// TIA Portal V16 export
// export: Created 2022-11-17T11:55:06.396Z, ExportSetting WithDefaults, DisplayName Totally Integrated Automation Portal, DisplayVersion V16 Update 6, DisplayName TIA Portal Version Control Interface, DisplayVersion V16 Update 2, DisplayName TIA Portal Openness, DisplayVersion V16 Update 6, DisplayName SINAMICS Startdrive Advanced, DisplayVersion V16 Update 5, DisplayName SINAMICS Startdrive G130, G150, S120, S150, SINAMICS MV, S210, DisplayVersion V16 Update 5, DisplayName SINAMICS Startdrive G110M, G120, G120C, G120D, G120P, G115D, DisplayVersion V16 Update 5, DisplayName STEP 7 Professional, DisplayVersion V16 Update 6, DisplayName STEP 7 Safety, DisplayVersion V16, DisplayName WinCC Advanced, DisplayVersion V16 Update 6
FUNCTION "FC11_PressureRectangularPn5W" : Void   // FC11, LAD
{ S7_Optimized_Access := 'FALSE' }
VERSION : 0.1
// stored: AutoNumber false, IsIECCheckEnabled false, SetENOAutomatically false, UDAEnableTagReadback false
BEGIN

REGION Network 1: Timeout for pressure plate upward/downward
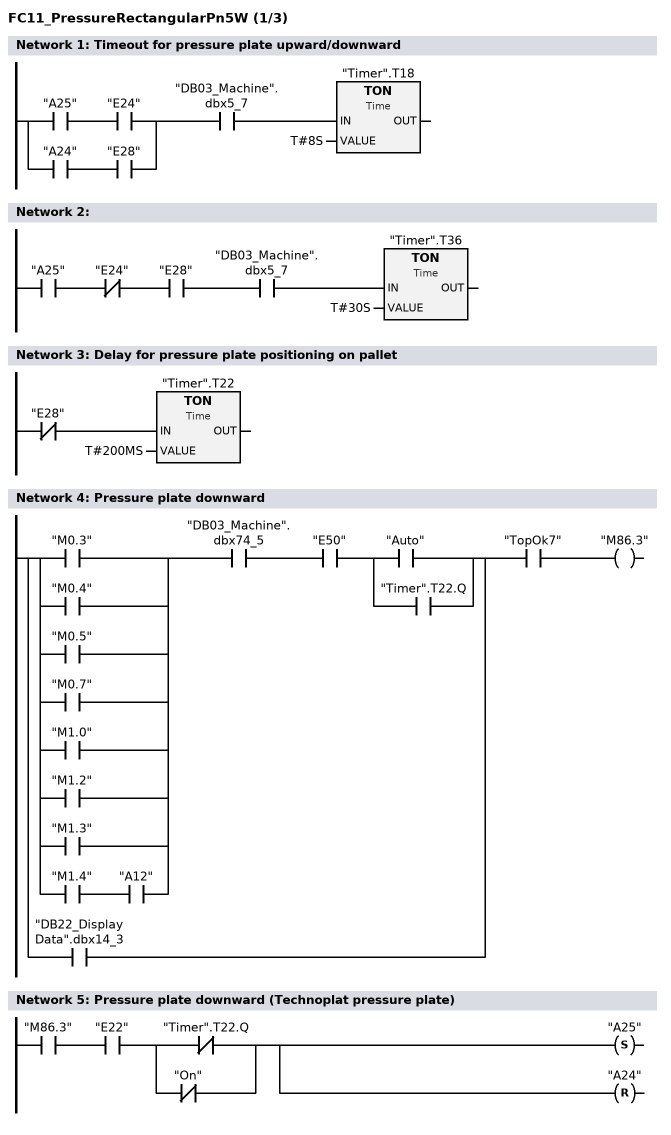
   "Timer".T18.TON(IN := (("A25" AND "E24") OR ("A24" AND "E28")) AND "DB03_Machine".dbx5_7, PT := T#8S);   // TON coil
END_REGION

REGION Network 2
   "Timer".T36.TON(IN := "A25" AND NOT "E24" AND "E28" AND "DB03_Machine".dbx5_7, PT := T#30S);   // TON coil
END_REGION

REGION Network 3: Delay for pressure plate positioning on pallet
   "Timer".T22.TON(IN := NOT "E28", PT := T#200MS);   // TON coil
END_REGION

REGION Network 4: Pressure plate downward
   RUNG wire#powerrail
      Contact( "M0.3" )
      wire#w1
      Contact( "DB03_Machine".dbx74_5 )
      Contact( "E50" )
      wire#w2
      Contact( "Auto" )
      wire#w3
      Contact( "TopOk7" )
      Coil( "M86.3" )
   END_RUNG
   RUNG wire#powerrail
      Contact( "M0.4" )
   END_RUNG wire#w1
   RUNG wire#powerrail
      Contact( "M0.5" )
   END_RUNG wire#w1
   RUNG wire#powerrail
      Contact( "M0.7" )
   END_RUNG wire#w1
   RUNG wire#powerrail
      Contact( "M1.0" )
   END_RUNG wire#w1
   RUNG wire#powerrail
      Contact( "M1.2" )
   END_RUNG wire#w1
   RUNG wire#powerrail
      Contact( "M1.3" )
   END_RUNG wire#w1
   RUNG wire#powerrail
      Contact( "M1.4" )
      Contact( "A12" )
   END_RUNG wire#w1
   RUNG wire#w2
      Contact( "Timer".T22.Q )
   END_RUNG wire#w3
   RUNG wire#powerrail
      Contact( "DB22_DisplayData".dbx14_3 )
   END_RUNG wire#w3
   // the same network as SCL:
   "M86.3" := ((("M0.3" OR "M0.4" OR "M0.5" OR "M0.7" OR "M1.0" OR "M1.2" OR "M1.3" OR ("M1.4" AND "A12")) AND "DB03_Machine".dbx74_5 AND "E50" AND ("Auto" OR "Timer".T22.Q)) OR "DB22_DisplayData".dbx14_3) AND "TopOk7";
END_REGION

REGION Network 5: Pressure plate downward (Technoplat pressure plate)
   RUNG wire#powerrail
      Contact( "M86.3" )
      Contact( "E22" )
      wire#w1
      I_Contact( "Timer".T22.Q )
      wire#w2
      S_Coil( "A25" )
   END_RUNG
   RUNG wire#w1
      I_Contact( "On" )
   END_RUNG wire#w2
   RUNG wire#w2
      R_Coil( "A24" )
   END_RUNG
   // the same network as SCL:
   IF "M86.3" AND "E22" AND (NOT "Timer".T22.Q OR NOT "On") THEN
       "A25" := TRUE;
       "A24" := FALSE;
   END_IF;
END_REGION

REGION Network 6: Pressure plate upward
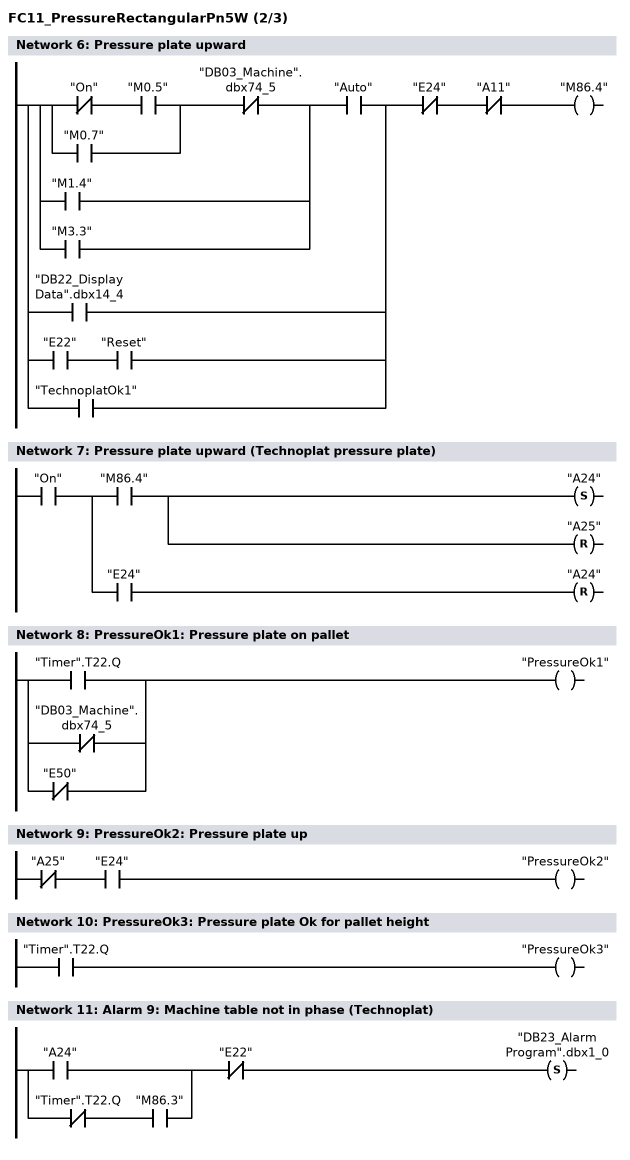
   RUNG wire#powerrail
      I_Contact( "On" )
      Contact( "M0.5" )
      wire#w1
      I_Contact( "DB03_Machine".dbx74_5 )
      wire#w2
      Contact( "Auto" )
      wire#w3
      I_Contact( "E24" )
      I_Contact( "A11" )
      Coil( "M86.4" )
   END_RUNG
   RUNG wire#powerrail
      Contact( "M0.7" )
   END_RUNG wire#w1
   RUNG wire#powerrail
      Contact( "M1.4" )
   END_RUNG wire#w2
   RUNG wire#powerrail
      Contact( "M3.3" )
   END_RUNG wire#w2
   RUNG wire#powerrail
      Contact( "DB22_DisplayData".dbx14_4 )
   END_RUNG wire#w3
   RUNG wire#powerrail
      Contact( "E22" )
      Contact( "Reset" )
   END_RUNG wire#w3
   RUNG wire#powerrail
      Contact( "TechnoplatOk1" )
   END_RUNG wire#w3
   // the same network as SCL:
   "M86.4" := ((((((NOT "On" AND "M0.5") OR "M0.7") AND NOT "DB03_Machine".dbx74_5) OR "M1.4" OR "M3.3") AND "Auto") OR "DB22_DisplayData".dbx14_4 OR ("E22" AND "Reset") OR "TechnoplatOk1") AND NOT "E24" AND NOT "A11";
END_REGION

REGION Network 7: Pressure plate upward (Technoplat pressure plate)
   RUNG wire#powerrail
      Contact( "On" )
      wire#w1
      Contact( "M86.4" )
      wire#w2
      S_Coil( "A24" )
   END_RUNG
   RUNG wire#w2
      R_Coil( "A25" )
   END_RUNG
   RUNG wire#w1
      Contact( "E24" )
      R_Coil( "A24" )
   END_RUNG
   // the same network as SCL:
   IF "On" AND "M86.4" THEN
       "A24" := TRUE;
       "A25" := FALSE;
   END_IF;
   IF "On" AND "E24" THEN "A24" := FALSE; END_IF;
END_REGION

REGION Network 8: PressureOk1: Pressure plate on pallet
   RUNG wire#powerrail
      Contact( "Timer".T22.Q )
      wire#w1
      Coil( "PressureOk1" )
   END_RUNG
   RUNG wire#powerrail
      I_Contact( "DB03_Machine".dbx74_5 )
   END_RUNG wire#w1
   RUNG wire#powerrail
      I_Contact( "E50" )
   END_RUNG wire#w1
   // the same network as SCL:
   "PressureOk1" := "Timer".T22.Q OR NOT "DB03_Machine".dbx74_5 OR NOT "E50";
END_REGION

REGION Network 9: PressureOk2: Pressure plate up
   RUNG wire#powerrail
      I_Contact( "A25" )
      Contact( "E24" )
      Coil( "PressureOk2" )
   END_RUNG
   // the same network as SCL:
   "PressureOk2" := NOT "A25" AND "E24";
END_REGION

REGION Network 10: PressureOk3: Pressure plate Ok for pallet height
   RUNG wire#powerrail
      Contact( "Timer".T22.Q )
      Coil( "PressureOk3" )
   END_RUNG
   // the same network as SCL:
   "PressureOk3" := "Timer".T22.Q;
END_REGION

REGION Network 11: Alarm 9: Machine table not in phase (Technoplat)
   RUNG wire#powerrail
      Contact( "A24" )
      wire#w1
      I_Contact( "E22" )
      S_Coil( "DB23_AlarmProgram".dbx1_0 )
   END_RUNG
   RUNG wire#powerrail
      I_Contact( "Timer".T22.Q )
      Contact( "M86.3" )
   END_RUNG wire#w1
   // the same network as SCL:
   IF ("A24" OR (NOT "Timer".T22.Q AND "M86.3")) AND NOT "E22" THEN
       "DB23_AlarmProgram".dbx1_0 := TRUE;
   END_IF;
END_REGION

REGION Network 12: Alarm 15: Pressure plate not up (Pressure plate)
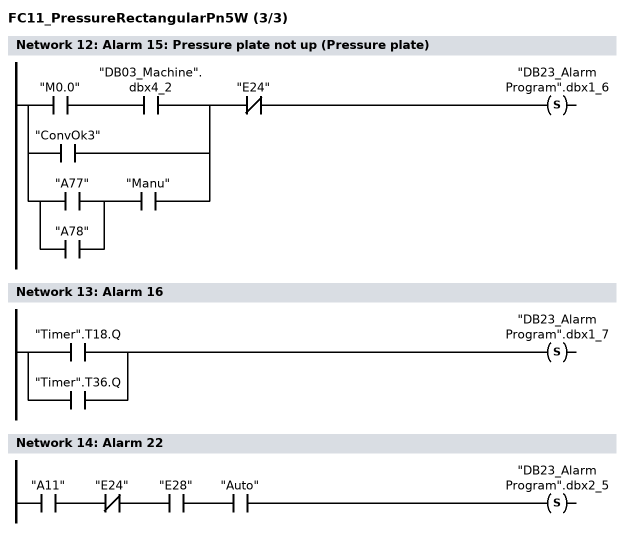
   RUNG wire#powerrail
      Contact( "M0.0" )
      Contact( "DB03_Machine".dbx4_2 )
      wire#w1
      I_Contact( "E24" )
      S_Coil( "DB23_AlarmProgram".dbx1_6 )
   END_RUNG
   RUNG wire#powerrail
      Contact( "ConvOk3" )
   END_RUNG wire#w1
   RUNG wire#powerrail
      Contact( "A77" )
      wire#w2
      Contact( "Manu" )
   END_RUNG wire#w1
   RUNG wire#powerrail
      Contact( "A78" )
   END_RUNG wire#w2
   // the same network as SCL:
   IF (("M0.0" AND "DB03_Machine".dbx4_2) OR "ConvOk3" OR (("A77" OR "A78") AND "Manu")) AND NOT "E24" THEN
       "DB23_AlarmProgram".dbx1_6 := TRUE;
   END_IF;
END_REGION

REGION Network 13: Alarm 16
   RUNG wire#powerrail
      Contact( "Timer".T18.Q )
      wire#w1
      S_Coil( "DB23_AlarmProgram".dbx1_7 )
   END_RUNG
   RUNG wire#powerrail
      Contact( "Timer".T36.Q )
   END_RUNG wire#w1
   // the same network as SCL:
   IF "Timer".T18.Q OR "Timer".T36.Q THEN "DB23_AlarmProgram".dbx1_7 := TRUE; END_IF;
END_REGION

REGION Network 14: Alarm 22
   RUNG wire#powerrail
      Contact( "A11" )
      I_Contact( "E24" )
      Contact( "E28" )
      Contact( "Auto" )
      S_Coil( "DB23_AlarmProgram".dbx2_5 )
   END_RUNG
   // the same network as SCL:
   IF "A11" AND NOT "E24" AND "E28" AND "Auto" THEN "DB23_AlarmProgram".dbx2_5 := TRUE; END_IF;
END_REGION
END_FUNCTION
